FUNCTION_BLOCK basicHorimetro (* Basic Function Block Type *)
  (* Standard: 61499-2 *)
  (* Version 0.0, 13/01/2026, Schneider Electric, Template *)
  PACKAGE Hidryco.HidrycoLib;
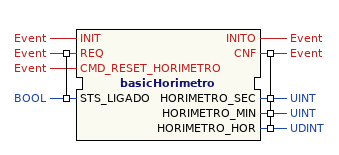
  EVENT_INPUT
    INIT; (* Initialization Request *)
    REQ WITH STS_LIGADO; (* Pulso 1S *)
    CMD_RESET_HORIMETRO;
  END_EVENT
  EVENT_OUTPUT
    INITO; (* Initialization Confirm *)
    CNF WITH HORIMETRO_SEC, HORIMETRO_MIN, HORIMETRO_HOR; (* Execution Confirmation *)
  END_EVENT
  VAR_INPUT
    STS_LIGADO : BOOL;
  END_VAR
  VAR_OUTPUT
    HORIMETRO_SEC : UINT;
    HORIMETRO_MIN : UINT;
    HORIMETRO_HOR : UDINT;
  END_VAR
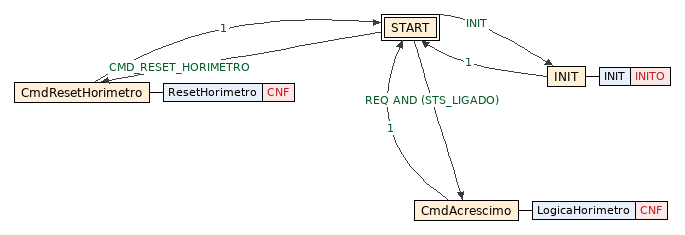
  EC_STATES
    START; (* Initial State *)
    INIT : INIT -> INITO; (* Initialization *)
    CmdAcrescimo : LogicaHorimetro -> CNF;
    CmdResetHorimetro : ResetHorimetro -> CNF;
  END_STATES
  EC_TRANSITIONS
    START TO INIT := INIT;
    INIT TO START := 1;
    START TO CmdAcrescimo := REQ AND (STS_LIGADO);
    CmdAcrescimo TO START := 1;
    START TO CmdResetHorimetro := CMD_RESET_HORIMETRO;
    CmdResetHorimetro TO START := 1;
  END_TRANSITIONS
  ALGORITHM INIT IN ST: (* Initialization algorithm *)
;
  END_ALGORITHM
  ALGORITHM REQ IN ST: (* Normally executed algorithm *)
;
  END_ALGORITHM
  ALGORITHM LogicaHorimetro IN ST:
// Incrementa segundos se houver pulso de 1 segundo e o equipamento estiver ligado
HORIMETRO_SEC := HORIMETRO_SEC + 1;

// Incrementa minutos e reseta segundos se os segundos ultrapassarem 59
IF (HORIMETRO_SEC > 59) THEN
	HORIMETRO_MIN := HORIMETRO_MIN + 1;
	HORIMETRO_SEC := 0;
END_IF;

// Incrementa horas e reseta minutos se os minutos ultrapassarem 59
IF (HORIMETRO_MIN > 59) THEN
    HORIMETRO_HOR := HORIMETRO_HOR + 1;
    HORIMETRO_MIN := 0;
END_IF;
  END_ALGORITHM
  ALGORITHM ResetHorimetro IN ST:
HORIMETRO_SEC := 0;
HORIMETRO_MIN := 0;
HORIMETRO_HOR := 0;
;
  END_ALGORITHM
END_FUNCTION_BLOCK
